{attribute 'qualified_only'}
VAR_GLOBAL
	DI_BtnYellow 	AT %I* : BOOL;
	DO_LampRed 		AT %Q* : BOOL;
	DO_LampGreen	AT %Q* : BOOL;
END_VAR

(* stored: Version 1.1.0.1, ProductVersion 3.1.4024.9
   GVL GVL_IO: Id {69f73459-75c2-4af2-ba4e-a6e34bb922db} *)
